VAR_GLOBAL
    g_iSizeOfGGOArray : INT := 50;

    g_stSystem	:	ST_System(*System_Struct*):= (
        xFirstScan := TRUE
    );

    g_DummyVG	:	ST_VG;


     fbGetCurTaskIdx : GETCURTASKINDEX;
     TaskInfo:PlcTaskSystemInfo;


END_VAR

(* stored: Version 1.1.0.1, ProductVersion 3.1.4022.18
   GVL Global_Variables: Id {a6c265d3-24f0-4c94-8227-7e6ead61f239} *)
